FUNCTION_BLOCK Crane
VAR_INPUT
	InputReady : BOOL;
	CraneDownSensor : BOOL;
	CraneUpSensor : BOOL;
	CraneAboveInput : BOOL;
	CraneAboveOutput : BOOL;
	InputSensor: BOOL;
	OutputSensor: BOOL;
	LoadReady: BOOL;
	LoadGrabbed: BOOL;
	CraneIsUp: BOOL;
	CraneIsDown : BOOL;
	HoldingItem: BOOL;
END_VAR
VAR_OUTPUT
	//right is down left is up
	HorizontalMotor : MOD_Crane_stMotorOutput;
	VerticalMotor : MOD_Crane_stMotorOutput;
	Grab : BOOL;
END_VAR
VAR
	State: INT;
	MotorDirection : (Left, Right, Stopped);

	
END_VAR

CASE State OF
	10://startup //reset?

		
		
	20://check box ready
		//wait untill
		IF InputReady = TRUE THEN
			State := 30;
		END_IF
	
	30://move crane down
		
		VerticalMotor.MoveLeft := TRUE;
		VerticalMotor.MoveRight := FALSE;
		
		IF CraneDownSensor = TRUE THEN
			State := 40;
		END_IF
		
	40://grab the load
		VerticalMotor.MoveLeft := FALSE;
		VerticalMotor.MoveRight := FALSE;
		Grab := TRUE;
		
		IF LoadGrabbed = TRUE THEN
			State := 50;
		END_IF

	50://move crane up
		VerticalMotor.MoveLeft := TRUE;
		VerticalMotor.MoveRight := FALSE;
		Grab := TRUE;
		
		IF CraneUpSensor = TRUE THEN
			State := 60;
		END_IF

	60://move crane to output position
		VerticalMotor.MoveLeft := FALSE;
		VerticalMotor.MoveRight := FALSE;
		HorizontalMotor.MoveLeft := TRUE;
		HorizontalMotor.MoveRight := FALSE;
		Grab := TRUE;
		IF CraneAboveInput = TRUE THEN
			State := 70;
		END_IF

	70://move crane down
		VerticalMotor.MoveLeft := FALSE;
		VerticalMotor.MoveRight := TRUE;
		HorizontalMotor.MoveLeft := FALSE;
		HorizontalMotor.MoveRight := FALSE;		
		IF OutputSensor = FALSE THEN
			State := 80;
		END_IF

	80://release load
		Grab := FALSE;
		IF HoldingItem = FALSE THEN
			State := 90;
		END_IF

	90://move crane up
		VerticalMotor.MoveLeft := TRUE;
		VerticalMotor.MoveRight := FALSE;
		HorizontalMotor.MoveLeft := FALSE;
		HorizontalMotor.MoveRight := FALSE;			
		IF CraneIsUp = TRUE THEN
			State := 100;
		END_IF	

	100://move crane over input
		VerticalMotor.MoveLeft := FALSE;
		VerticalMotor.MoveRight := FALSE;
		HorizontalMotor.MoveLeft := FALSE;
		HorizontalMotor.MoveRight := TRUE;			
		IF CraneAboveInput = TRUE THEN
			State := 20;
		END_IF

END_FUNCTION_BLOCK

(* stored: Version 1.1.0.1, ProductVersion 3.1.4024.6
   POU Crane: Id {5ef12530-d6be-413c-8970-2208adcc7e82}, SpecialFunc None *)
